// TIA Portal V19 export
DATA_BLOCK "MODULES_CTRL"   // DB54
{ S7_Optimized_Access := 'TRUE' }
// stored: MemoryReserve 100
   VAR
      ADIN { ExternalAccessible := 'False'; ExternalVisible := 'False'; ExternalWritable := 'False'; S7_SetPoint := 'True'} : Array[0.."M_ADIN"] of "CTRL_ADIN";
      AIN { ExternalAccessible := 'False'; ExternalVisible := 'False'; ExternalWritable := 'False'; S7_SetPoint := 'True'} : Array[0.."M_AIN"] of "CTRL_AIN";
      CVLV { ExternalAccessible := 'False'; ExternalVisible := 'False'; ExternalWritable := 'False'; S7_SetPoint := 'True'} : Array[0.."M_CVLV"] of "CTRL_CVLV";
      DIFF { ExternalAccessible := 'False'; ExternalVisible := 'False'; ExternalWritable := 'False'; S7_SetPoint := 'True'} : Array[0.."M_DIFF"] of "CTRL_DIFF";
      DIN { ExternalAccessible := 'False'; ExternalVisible := 'False'; ExternalWritable := 'False'; S7_SetPoint := 'True'} : Array[0.."M_DIN"] of "CTRL_DIN";
      MTRDIR { ExternalAccessible := 'False'; ExternalVisible := 'False'; ExternalWritable := 'False'; S7_SetPoint := 'True'} : Array[0.."M_MTRDIR"] of "CTRL_MTRDIR";
      MTRLIN { ExternalAccessible := 'False'; ExternalVisible := 'False'; ExternalWritable := 'False'; S7_SetPoint := 'True'} : Array[0.."M_MTRLIN"] of "CTRL_MTRLIN";
      MTR { ExternalAccessible := 'False'; ExternalVisible := 'False'; ExternalWritable := 'False'; S7_SetPoint := 'True'} : Array[0.."M_MTR"] of "CTRL_MTR";
      VLV { ExternalAccessible := 'False'; ExternalVisible := 'False'; ExternalWritable := 'False'; S7_SetPoint := 'True'} : Array[0.."M_VLV"] of "CTRL_VLV";
   END_VAR
BEGIN
END_DATA_BLOCK
